TYPE T_IdBaseSendData :
STRUCT
	fbDataChannel						: FB_IdBaseSendDch;
	rDataChannelItem					: T_IdBase_DCH;
	fbFifo								: FB_DataChannelSenderFifo;
END_STRUCT
END_TYPE

(* stored: Version 1.1.0.1, ProductVersion 3.1.0.24
   DUT T_IdBaseSendData: Id {d90f58cb-2ee6-4305-a3d8-23931ed538f9} *)
